# B&R Automation Studio project LR3
Automation Studio 

## Logical view

- Data object Logical/GmcIpUserConfig/gmcipvar (Cnc, version 5.02.1) (no source held here)

- Data object Logical/GmcIpUserConfig/gmcipusm (Cnc, version 5.02.1) (no source held here)

- Data object Logical/GmcIpUserConfig/gmcipui (Cnc, version 5.02.1) (no source held here)

- Data object Logical/GmcIpUserConfig/gmcipus (Cnc, version 5.02.1) (no source held here)

### Program Logical/SDCAxisCtrl_Z (ANSIC)

#### Main.c - Init, cyclic, exit code
```c
#include <bur/plctypes.h>

#ifdef _DEFAULT_INCLUDES
	#include <AsDefault.h>
#endif

void _INIT ProgramInit(void)
{
	//Устанваливаем типы SDC модулей
	AxisZ_HW.EncIf1_Typ = ncSDC_ENC16;
	AxisZ_HW.DiDoIf_Typ = ncSDC_DIDO;
	AxisZ_HW.DrvIf_Typ = ncSDC_DRVSERVO16;

	//Устанавливаем имена переменных
	strcpy(AxisZ_HW.EncIf1_Name, "AxisZ_EncIf");
	strcpy(AxisZ_HW.DrvIf_Name, "AxisZ_DrvIf");
	strcpy(AxisZ_HW.DiDoIf_Name, "AxisZ_DiDoIf");

	//Устанавливаем входы готовности и нормальной работы
	AxisZ_EncIf.iEncOK = 1;
	AxisZ_DrvIf.iDrvOK = 1;
	AxisZ_DrvIf.iStatusEnable = 1;
	AxisZ_DiDoIf.iDriveReady = 1;

	fb_controller.dt = 0.002;
	fb_controller.k_i = 0.16;
	fb_controller.k_p = 0.0064;
	fb_controller.max_abs_value = 24.0;

	pwm_period = 20;
}

void _CYCLIC ProgramCyclic(void)
{
	FB_Axis(&axis_Z);
	coil_pwm_value = coil_powered ? 32767 : 0;

	increase_counters();

	//Формирование показаний датчика

	AxisZ_EncIf.iActTime = (INT) AsIOTimeCyclicStart();
	AxisZ_EncIf.iActPos = axis_Z.counter;
	AxisZ_DiDoIf.iPosHwEnd = axis_Z.endswitch_a_reached;
	AxisZ_DiDoIf.iNegHwEnd = axis_Z.endswitch_b_reached;
	fb_controller.in = AxisZ_DrvIf.oSetPos;

	if((fb_controller.in<min_task)&&(fb_controller.in>(-min_task))) fb_controller.in = 0;
	fb_controller.in = fb_controller.in * 6500/32767 - axis_Z.speed;

	FB_Controller(&fb_controller);

	axis_Z.pwm_value = fb_controller.out / 24.0 * 32767;

}

void increase_counters(void)
{
	AxisZ_EncIf.iLifeCnt++;
	AxisZ_DiDoIf.iLifeCntDriveEnable++;
	AxisZ_DiDoIf.iLifeCntDriveReady++;
	AxisZ_DiDoIf.iLifeCntNegHwEnd++;
	AxisZ_DiDoIf.iLifeCntPosHwEnd++;
	AxisZ_DiDoIf.iLifeCntReference++;
	AxisZ_DrvIf.iLifeCnt++;
}

void _EXIT ProgramExit(void)
{
	// Insert code here

}
```

- Visualisation Logical/Visu (not shown)

### Program Logical/User_Interface (ANSIC)

#### Variables.var
```iecst
VAR
	homing : MC_Home := (0);
	power : MC_Power := (0);
END_VAR
```

#### Main.c
```c
#include <bur/plctypes.h>

#ifdef _DEFAULT_INCLUDES
	#include <AsDefault.h>
#endif

void _INIT ProgramInit(void)
{
	// Объявление осей Y и Z по адресу
	Trajectory.AxisY = &AxisY;
	Trajectory.AxisZ = &AxisZ;

	// Мнгновенное присваивание значения 0 при инициализации переменной
	Trajectory.length = 0;
	Move_axis.length = 0;
}

void _CYCLIC ProgramCyclic(void)
{
	FB_Trajectory(&Trajectory); // Инициализация функционального блока
}

void _EXIT ProgramExit(void)
{

}
```

Listed in the project but not available here: Logical/Global.typ, Logical/Global.var, Logical/Libraries, Logical/Types.typ, Logical/AxisApt, Logical/AxisInit, Logical/acp10etxen, Logical/ncsdcctrl, Logical/gAxis03obj, Logical/GmcIpConfig, Logical/GmcIpUserConfig/gmcipfun, Logical/GmcIpUserConfig/gmcipfub, Logical/GmcIpUserConfig/gmcipubr, Logical/GmcIpUserConfig/gmcipuc, Logical/CncInit, Logical/CncProg, Logical/SDCAxisCtrl_X, Logical/SDCAxisCtrl_Y, Logical/SDCAxisCtrl_Z/Variables.var, Logical/CncProg1
